FUNCTION TryConvert_LREAL_TO_DT : BOOL
VAR_INPUT
	in : LREAL;
	out : REFERENCE TO DT;
END_VAR

IF in > DatatypeLimits.MAX_VALUE_OF_LREAL_WHICH_CAN_BE_HELD_IN_A_DT THEN
	RETURN;
END_IF

IF in < DatatypeLimits.MIN_VALUE_OF_LREAL_WHICH_CAN_BE_HELD_IN_A_DT THEN
	RETURN;
END_IF

out := LREAL_TO_DT(in);
TryConvert_LREAL_TO_DT := TRUE;

END_FUNCTION

(* stored: Version 1.1.0.1, ProductVersion 3.1.4024.12
   POU TryConvert_LREAL_TO_DT: Id {1fc115da-49dc-4292-819c-c1ec308e9841}, SpecialFunc None *)
